// TIA Portal V17 export
// export: Created 2022-12-08T07:31:26.4680568Z, ExportSetting WithDefaults, DisplayName Totally Integrated Automation Portal, DisplayVersion V17 Update 5, DisplayName TIA Portal Openness, DisplayVersion V17 Update 5, DisplayName TIA Portal Version Control Interface, DisplayVersion V17, DisplayName Simotion SCOUT TIA, DisplayVersion 5.4.3.0, DisplayName SINAMICS Startdrive Advanced, DisplayVersion V17 SP1, DisplayName SINAMICS Startdrive G130, G150, S120, S150, SINAMICS MV, S210, DisplayVersion V17 SP1, DisplayName SINAMICS Startdrive G110M, G120, G120C, G120D, G120P, G115D, DisplayVersion V17 SP1, DisplayName STEP 7 Professional, DisplayVersion V17 Update 5, DisplayName STEP 7 Safety, DisplayVersion V17, DisplayName WinCC Advanced, DisplayVersion V17 Update 5
DATA_BLOCK "DB_ProductionData"   // DB107
AUTHOR : EconoPak GmbH
VERSION : 0.1
// stored: AutoNumber false, DBAccessibleFromOPCUA true, DBAccessibleFromWebserver true, InstanceOfName FB_ProductionData, InstanceOfType FB
"FB_ProductionData"
   // VAR_INPUT
   //    i_Count1 : Bool;
   //    i_Count2 : Bool;
   //    i_Count3 : Bool;
   //    i_Count4 : Bool;
   //    i_CountNOK : Bool;
   //    i_ResetCounter : Bool;
   // END_VAR
   // VAR_IN_OUT
   //    iq_TotalOK : DInt;
   //    iq_TotalNOK : DInt;
   //    iq_Total : DInt;
   //    iq_CurrentMinute : DInt;
   //    iq_LastMinute : DInt;
   //    iq_CurrentHour : DInt;
   //    iq_LastHour : DInt;
   // END_VAR
   // VAR
   //    inst_Rtrig_Count1 : R_TRIG;
   //    inst_Rtrig_Count2 : R_TRIG;
   //    inst_Rtrig_Count3 : R_TRIG;
   //    inst_Rtrig_Count4 : R_TRIG;
   //    inst_Rtrig_CountNOK : R_TRIG;
   //    inst_Rtrig_OneMinute : R_TRIG;
   //    inst_Rtrig_OneHour : R_TRIG;
   //    inst_TON_Minute : TON_TIME;
   //    inst_TON_Hour : TON_TIME;
   // END_VAR
BEGIN
END_DATA_BLOCK
